PROGRAM MAIN
VAR
	fbPepPizza 	: FB_PepperoniPizza;
	fbVegPizza 	: FB_VeggiePizza;
	
	bPepButton: BOOL;
	bVegButton: BOOL;
END_VAR

fbPepPizza.makePizza(bPepButton);
fbVegPizza.makePizza(bVegButton);

END_PROGRAM

(* stored: Version 1.1.0.1, ProductVersion 3.1.4024.12
   POU MAIN: Id {c7c31f80-c7d0-4df9-9a94-06a2d4614184}, SpecialFunc None *)
